// TIA Portal V18 export
DATA_BLOCK "HMI DB"   // DB2
{ S7_Optimized_Access := 'FALSE' }
VERSION : 0.1
// stored: AutoNumber true, DBAccessibleFromOPCUA true, IsOnlyStoredInLoadMemory false, IsWriteProtectedInAS false
   VAR RETAIN
      "START PREP" : Bool := FALSE;
      "START CIP" : Bool := FALSE;
      "CIP 3 STEP" : Bool := FALSE;
      "CIP 5 STEP" : Bool := FALSE;
      "CIP 7 STEP" : Bool := FALSE;
      RP1 : Bool;
      RP2 : Bool;
      RP3 : Bool;
      "RESUME CIP" : Bool;
      "RP1 SELECTED" : Bool;
      "RP2 SELECTED" : Bool;
      "RP3 SELECTED" : Bool;
      "3 STEP STATUS" : Word;
      "5 STEP STATUS" : Word;
      "9 STEP STATUS" : Word;
      RESERVE : Array[0..28] of Word;
      "BFV1 AM" { S7_SetPoint := 'True'} : "AM CTRL";
      "BFV2 AM" { S7_SetPoint := 'True'} : "AM CTRL";
      "BFV3 AM" { S7_SetPoint := 'True'} : "AM CTRL";
      "BFV4 AM" { S7_SetPoint := 'True'} : "AM CTRL";
      "BFV5 AM" { S7_SetPoint := 'True'} : "AM CTRL";
      "BFV6 AM" { S7_SetPoint := 'True'} : "AM CTRL";
      "BFV7 AM" { S7_SetPoint := 'True'} : "AM CTRL";
      "BFV8 AM" { S7_SetPoint := 'True'} : "AM CTRL";
      "BFV9 AM" { S7_SetPoint := 'True'} : "AM CTRL";
      "BFV10 AM" { S7_SetPoint := 'True'} : "AM CTRL";
      "BFV11 AM" { S7_SetPoint := 'True'} : "AM CTRL";
      "BFV12 AM" { S7_SetPoint := 'True'} : "AM CTRL";
      "BFV13 AM" { S7_SetPoint := 'True'} : "AM CTRL";
      "BFV14 AM" { S7_SetPoint := 'True'} : "AM CTRL";
      "BFV15 AM" { S7_SetPoint := 'True'} : "AM CTRL";
      "BFV16 AM" { S7_SetPoint := 'True'} : "AM CTRL";
      "BFV17 AM" { S7_SetPoint := 'True'} : "AM CTRL";
      "BFV18 AM" { S7_SetPoint := 'True'} : "AM CTRL";
      "BFV19 AM" { S7_SetPoint := 'True'} : "AM CTRL";
      "VFD AM" { S7_SetPoint := 'True'} : "AM CTRL";
      "RETURN PUMP 1 AM" { S7_SetPoint := 'True'} : "AM CTRL";
      "RETURN PUMP 2 AM" { S7_SetPoint := 'True'} : "AM CTRL";
      "RETURN PUMP 3 AM" { S7_SetPoint := 'True'} : "AM CTRL";
      "CAUSTIC AM" { S7_SetPoint := 'True'} : "AM CTRL";
      "ACIDIC AM" { S7_SetPoint := 'True'} : "AM CTRL";
      "PUMP SLOW SP" : Int := 0;
      RECUP : "TANK DATA";
      "HOT WATER" : "TANK DATA";
      CAUSTIC : "TANK DATA";
      ACIDIC : "TANK DATA";
      "ANALOG VALUES" : Struct
         FLOW : Real := 0.0;
         CONDCTIVITY : Real := 0.0;
         "RECUP TEMP" : Real := 0.0;
         "HOT WTR TEMP" : Real := 0.0;
         "CAUSTIC TEMP" : Real := 0.0;
         "ACID TEMP" : Real := 0.0;
         "RETURN LINE TEMP" : Real := 0.0;
      END_STRUCT;
      "START DELAYS" : Struct
         "RP1 MIN" : Int;
         "RP1 SEC" : Int;
         "RP2 MIN" : Int;
         "RP2 SEC" : Int;
         "RP3 MIN" : Int;
         "RP3 SEC" : Int;
      END_STRUCT;
      "COMMON SETPOINTS" : Struct   // 286
         "COND MIN FOR RECUP" : Real;
         "TMP MIN FOR RECUP" : Real;
         "WATER FLUSH MIN" : Int;
         "WATER FLUSH SEC" : Int;
         "WATER FLUSH REM MIN" : Int;
         "WATER FLUSH REM SEC" : Int;
      END_STRUCT;
      "Fwd line temp" : Real;
   END_VAR
BEGIN
   "BFV1 AM"."AUTO/MAN" := TRUE;
   "BFV1 AM"."MAN START" := FALSE;
   "BFV1 AM"."MAN STOP" := FALSE;
   "BFV2 AM"."AUTO/MAN" := TRUE;
   "BFV2 AM"."MAN START" := FALSE;
   "BFV2 AM"."MAN STOP" := FALSE;
   "BFV3 AM"."AUTO/MAN" := TRUE;
   "BFV3 AM"."MAN START" := FALSE;
   "BFV3 AM"."MAN STOP" := FALSE;
   "BFV4 AM"."AUTO/MAN" := TRUE;
   "BFV4 AM"."MAN START" := FALSE;
   "BFV4 AM"."MAN STOP" := FALSE;
   "BFV5 AM"."AUTO/MAN" := TRUE;
   "BFV5 AM"."MAN START" := FALSE;
   "BFV5 AM"."MAN STOP" := FALSE;
   "BFV6 AM"."AUTO/MAN" := TRUE;
   "BFV6 AM"."MAN START" := FALSE;
   "BFV6 AM"."MAN STOP" := FALSE;
   "BFV7 AM"."AUTO/MAN" := TRUE;
   "BFV7 AM"."MAN START" := FALSE;
   "BFV7 AM"."MAN STOP" := FALSE;
   "BFV8 AM"."AUTO/MAN" := TRUE;
   "BFV8 AM"."MAN START" := FALSE;
   "BFV8 AM"."MAN STOP" := FALSE;
   "BFV9 AM"."AUTO/MAN" := TRUE;
   "BFV9 AM"."MAN START" := FALSE;
   "BFV9 AM"."MAN STOP" := FALSE;
   "BFV10 AM"."AUTO/MAN" := TRUE;
   "BFV10 AM"."MAN START" := FALSE;
   "BFV10 AM"."MAN STOP" := FALSE;
   "BFV11 AM"."AUTO/MAN" := TRUE;
   "BFV11 AM"."MAN START" := FALSE;
   "BFV11 AM"."MAN STOP" := FALSE;
   "BFV12 AM"."AUTO/MAN" := TRUE;
   "BFV12 AM"."MAN START" := FALSE;
   "BFV12 AM"."MAN STOP" := FALSE;
   "BFV13 AM"."AUTO/MAN" := TRUE;
   "BFV13 AM"."MAN START" := FALSE;
   "BFV13 AM"."MAN STOP" := FALSE;
   "BFV14 AM"."AUTO/MAN" := TRUE;
   "BFV14 AM"."MAN START" := FALSE;
   "BFV14 AM"."MAN STOP" := FALSE;
   "BFV15 AM"."AUTO/MAN" := TRUE;
   "BFV15 AM"."MAN START" := FALSE;
   "BFV15 AM"."MAN STOP" := FALSE;
   "BFV16 AM"."AUTO/MAN" := TRUE;
   "BFV16 AM"."MAN START" := FALSE;
   "BFV16 AM"."MAN STOP" := FALSE;
   "BFV17 AM"."AUTO/MAN" := TRUE;
   "BFV17 AM"."MAN START" := FALSE;
   "BFV17 AM"."MAN STOP" := FALSE;
   "BFV18 AM"."AUTO/MAN" := TRUE;
   "BFV18 AM"."MAN START" := FALSE;
   "BFV18 AM"."MAN STOP" := FALSE;
   "BFV19 AM"."AUTO/MAN" := TRUE;
   "BFV19 AM"."MAN START" := FALSE;
   "BFV19 AM"."MAN STOP" := FALSE;
   "VFD AM"."AUTO/MAN" := TRUE;
   "VFD AM"."MAN START" := FALSE;
   "VFD AM"."MAN STOP" := FALSE;
   "RETURN PUMP 1 AM"."AUTO/MAN" := TRUE;
   "RETURN PUMP 1 AM"."MAN START" := FALSE;
   "RETURN PUMP 1 AM"."MAN STOP" := FALSE;
   "RETURN PUMP 2 AM"."AUTO/MAN" := TRUE;
   "RETURN PUMP 2 AM"."MAN START" := FALSE;
   "RETURN PUMP 2 AM"."MAN STOP" := FALSE;
   "RETURN PUMP 3 AM"."AUTO/MAN" := TRUE;
   "RETURN PUMP 3 AM"."MAN START" := FALSE;
   "RETURN PUMP 3 AM"."MAN STOP" := FALSE;
   "CAUSTIC AM"."AUTO/MAN" := TRUE;
   "CAUSTIC AM"."MAN START" := FALSE;
   "CAUSTIC AM"."MAN STOP" := FALSE;
   "ACIDIC AM"."AUTO/MAN" := TRUE;
   "ACIDIC AM"."MAN START" := FALSE;
   "ACIDIC AM"."MAN STOP" := FALSE;
   RECUP."COND SP" := 0.0;
   RECUP."HYSTERIRIS TEMP" := 0.0;
   RECUP."HYSTERISIS COND" := 0.0;
   RECUP."CYCLE TIME SEC" := 0;
   RECUP."ELAPSED MIN" := 0;
   RECUP."ELAPSED SEC" := 0;
   "HOT WATER"."COND SP" := 0.0;
   "HOT WATER"."HYSTERIRIS TEMP" := 0.0;
   "HOT WATER"."HYSTERISIS COND" := 0.0;
   "HOT WATER"."CYCLE TIME MIN" := 0;
   "HOT WATER"."CYCLE TIME SEC" := 0;
   "HOT WATER"."ELAPSED MIN" := 0;
   "HOT WATER"."ELAPSED SEC" := 0;
   CAUSTIC."COND SP" := 0.0;
   CAUSTIC."HYSTERIRIS TEMP" := 0.0;
   CAUSTIC."HYSTERISIS COND" := 0.0;
   CAUSTIC."CYCLE TIME MIN" := 0;
   CAUSTIC."CYCLE TIME SEC" := 0;
   CAUSTIC."ELAPSED MIN" := 0;
   CAUSTIC."ELAPSED SEC" := 0;
   ACIDIC."COND SP" := 0.0;
   ACIDIC."HYSTERIRIS TEMP" := 0.0;
   ACIDIC."HYSTERISIS COND" := 0.0;
   ACIDIC."CYCLE TIME MIN" := 0;
   ACIDIC."CYCLE TIME SEC" := 0;
   ACIDIC."ELAPSED MIN" := 0;
   ACIDIC."ELAPSED SEC" := 0;
END_DATA_BLOCK
